// TIA Portal V17 export
// export: Created 2024-06-19T09:47:14.1555743Z, ExportSetting WithDefaults, DisplayName Totally Integrated Automation Portal, DisplayVersion V17, DisplayName TIA Portal Openness, DisplayVersion V17, DisplayName TIA Portal Version Control Interface, DisplayVersion V17, DisplayName STEP 7 Professional, DisplayVersion V17, DisplayName STEP 7 Safety, DisplayVersion V17, DisplayName WinCC Professional, DisplayVersion V17
DATA_BLOCK "St0_Out"   // DB15
{ S7_Optimized_Access := 'TRUE' }
VERSION : 0.1
// stored: AutoNumber false, DBAccessibleFromOPCUA true, DBAccessibleFromWebserver true, IsOnlyStoredInLoadMemory false, IsRetainMemResEnabled false, IsWriteProtectedInAS false, MemoryReserve 100
   VAR
      Verrou_PorteEntree : Bool;
      Verrou_PorteSortie : Bool;
      Verrou_PorteVision : Bool;
      Verrou_PorteArriere : Bool;
      Ouverture_PorteEntree : Bool;
      Ouverture_PorteSortie : Bool;
      LED_Rouge : Bool;
      LED_Orange : Bool;
      LED_Vert : Bool;
      LED_Bleu : Bool;
   END_VAR
BEGIN
END_DATA_BLOCK
